INTERFACE PUBLIC I_DigitalOutput EXTENDS __System.IQueryInterface

{attribute 'monitoring' := 'call'}
PROPERTY PUBLIC State : BOOL
GET
END_GET
SET
END_SET
END_PROPERTY

END_INTERFACE

(* stored: Version 1.1.0.1, ProductVersion 3.1.4024.12
   Itf I_DigitalOutput: Id {283a026b-1a0b-4fd4-a19f-634c7ddd0eca}
   Property State: Id {97c1f9c5-3b25-485c-8b62-5328d54a2c65}
   Get Get: Id {83e6df0c-b157-4066-bb8d-361ea78d1869}
   Set Set: Id {81b54612-c219-4b5c-9341-ba0ac862b065} *)
